PROGRAM MAIN
VAR
	cleanin: fb_cleanIn;
	cleanout: fb_cleanOut;
	undock: fb_undock;
	dock: fb_dock;
	switchclk: fb_switchclkcheck;
	opcl: fb_dsopenclose;
	allundock: fb_engageUndockAll;
	alldock: fb_engageDockAll;
	stop : TC_Stop;
	pisttest: fb_testpiston;
END_VAR

(*always running*)

IF TCin.toolOn THEN
	switchclk();
END_IF

(*engaged manually*)
IF engage.stepper THEN
	opcl();
END_IF

IF engage.cleanIn THEN
	cntrlstate.cleanin := FALSE;
	cleanin(done := cntrlstate.cleanin);
	IF cntrlstate.cleanin THEN
		engage.cleanIn := FALSE;
	END_IF
END_IF

IF engage.cleanOut THEN
	cntrlstate.cleanout := FALSE;
	cleanout(done := cntrlstate.cleanout);
	IF cntrlstate.cleanout THEN
		engage.cleanOut := FALSE;
	END_IF
END_IF

IF engage.undock THEN
	cntrlstate.undock := FALSE;
	undock();
	IF cntrlstate.undock THEN
		engage.undock := FALSE;
	END_IF
END_IF

IF engage.dock THEN
	cntrlstate.dock := FALSE;
	dock(toolID := 4);
	IF cntrlstate.dock THEN
		engage.dock := FALSE;
	END_IF
END_IF


(*engage a sequence*)
IF engage.allundock THEN
	allundock();
END_IF

IF engage.alldock THEN
	alldock();
END_IF

(*errorHandle stopping plc*)
IF NOT switchclk.swXgood THEN
	stop(STOP:=TRUE);
END_IF


(*TESTING*)
IF engage.pisttest THEN
	pisttest();
END_IF

END_PROGRAM

(* stored: Version 1.1.0.1, ProductVersion 3.1.4024.5
   POU MAIN: Id {eb432b23-e1d0-434b-99f7-8e0d8288ae20}, SpecialFunc None *)
